{attribute 'qualified_only'}
{attribute 'strict'}
TYPE PointMode :
(
	notUsed		:= -1,
	docking 	:= 1,
	transfer	:= 2
);
END_TYPE

(* stored: Version 1.1.0.1, ProductVersion 3.1.4024.11
   DUT PointMode: Id {0365e72b-1c56-494e-8508-358ecd299222} *)
